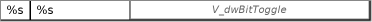
VISUALIZATION V_LiquidSensorCfg  // 372x22
VAR_INPUT
  iNumOfCh : INT;
END_VAR
VAR_IN_OUT
	IOfbLiquidSensor : FB_LiquidSensor;
END_VAR
    Rectangle (130,0 240x20)
    Rectangle (0,0 30x20), "%s", text variable: IOfbLiquidSensor.iChan
    Rectangle (30,0 100x20), "%s", text variable: IOfbLiquidSensor.VnvszName
        OnMouseDown: write the text variable via Default
    Frame (130,0 239x19)
        shows V_dwBitToggle(iNumOfCh := iNumOfCh, dwVar := IOfbLiquidSensor.VnvdwCFGLiquidToTransor)
END_VISUALIZATION

(* stored: Version 1.1.0.1, ProductVersion 3.1.4018.10
   Visu V_LiquidSensorCfg: Id {7ad6b34f-2dde-4819-9a80-35d26b074307} *)
